{attribute 'GeneratedUsingTerminal: EL2522-0000-0017'}
{attribute addProperty BoxType "EL2522-0000-0017"}
{attribute addProperty Id "ControlAT %Q*Control_DAEE1D523Frequency_valueAT %Q*UINT2"}
{attribute addProperty CRC "2458384612"}
{attribute addProperty Size "5"}
TYPE PTO_Control_Channel_9287F8E4 :
STRUCT
	{attribute addProperty Name "Control"}
	Control AT %Q* : Control_DAEE1D52;
	{attribute addProperty Name "Frequency_value"}
	Frequency_value AT %Q* : UINT;
END_STRUCT
END_TYPE

(* stored: Version 1.2.0.0, ProductVersion 3.1.4024.9
   DUT PTO_Control_Channel_9287F8E4: Id {d3fb87b2-1dfc-443b-9ffd-9a04bd0d6a06} *)
